PROGRAM MAIN
VAR
	
END_VAR


IF GVL.apparaatLeeg THEN
	GVL.state := 1;
	GVL.allesLegen := FALSE;
	GVL.apparaatLeeg := FALSE;
END_IF

CASE state OF
	1: 				//Apparaat staat uit, de gebruiker kan het apparaat vullen
		IF GVL.allesLegen OR GVL.apparaatAanzetten THEN
			GVL.koffieError := TRUE;
		ELSE
			GVL.koffieError := FALSE;
		END_IF
		
		IF GVL.filterPlaatsen AND NOT GVL.filterGeplaatst THEN
			GVL.filterGeplaatst := TRUE;
		END_IF
		
		IF GVL.scoopieDrBij THEN
			GVL.aantalSchepjes := GVL.storeSchepjes + 1;
		ELSE
			GVL.storeSchepjes := GVL.aantalschepjes;
		END_IF
		
		IF GVL.waterreservoirVullen THEN
			GVL.reservoirLevel := GVL.storeReservoir + 1;
		ELSE
			GVL.storeReservoir := GVL.reservoirLevel;
		END_IF
		
		IF GVL.apparaatAanzetten THEN
			GVL.state := 2;
		END_IF
		
	2: 				//Apparaat staat aan, koffie wordt gezet op basis van de gebruikersinputs
		
		IF GVL.aantalSchepjes = 2*GVL.reservoirLevel THEN
			GVL.lekkereKoffie := TRUE;
		ELSIF GVL.aantalSchepjes < 2*GVL.reservoirLevel THEN
			GVL.waterigeKoffie := TRUE;
		ELSIF GVL.aantalSchepjes > 2*GVL.reservoirLevel THEN
			GVL.sterkeKoffie := TRUE;
		
			IF GVL.ikBenMoe THEN
				GVL.lekkereKoffie := TRUE;
			END_IF
			
		END_IF
		GVL.apparaatLeeg := FALSE;
		GVL.koffieKlaar := TRUE;
		
		IF GVL.allesLegen THEN
			resetVars();
		END_IF
		
END_CASE;

END_PROGRAM

(* stored: Version 1.1.0.1, ProductVersion 3.1.4024.12
   POU MAIN: Id {f5f2698f-4123-4600-9405-b57764ad172b}, SpecialFunc None *)
